FUNCTION_BLOCK MsgpParse (* Tamplate for a simple Basic Function Block Type *)
  (* Standard: 61499-2 *)
  (* Version 0.0, 2018-05-31, 4DIAC-IDE, 4DIAC-Consortium *)
  (* Version 1.0, 2016-05-26, AZ, fortiss GmbH *)
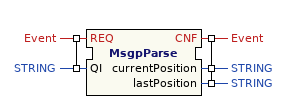
  EVENT_INPUT
    REQ WITH QI; (* Normal Execution Request *)
  END_EVENT
  EVENT_OUTPUT
    CNF WITH currentPosition, lastPosition; (* Execution Confirmation *)
  END_EVENT
  VAR_INPUT
    QI : STRING; (* Head+vechlie_currentPosition_LastPosition+end *)
  END_VAR
  VAR_OUTPUT
    currentPosition : STRING; (* position value 2 *)
    lastPosition : STRING; (* position value ,2 *)
  END_VAR
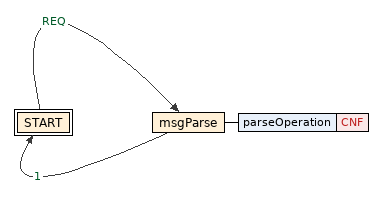
  EC_STATES
    START; (* Initial State *)
    msgParse : parseOperation -> CNF; (* Normal execution *)
  END_STATES
  EC_TRANSITIONS
    START TO msgParse := REQ;
    msgParse TO START := 1;
  END_TRANSITIONS
  ALGORITHM parseOperation IN ST: (* new algorithm *)
QI:='ok';
currentPosition:="12";
lastPosition :="22";
  END_ALGORITHM
END_FUNCTION_BLOCK
